// LS Electric XG5000 project: Master_UPH
// PLC LSPLC

PROGRAM NewProgram (task: Scan Program)

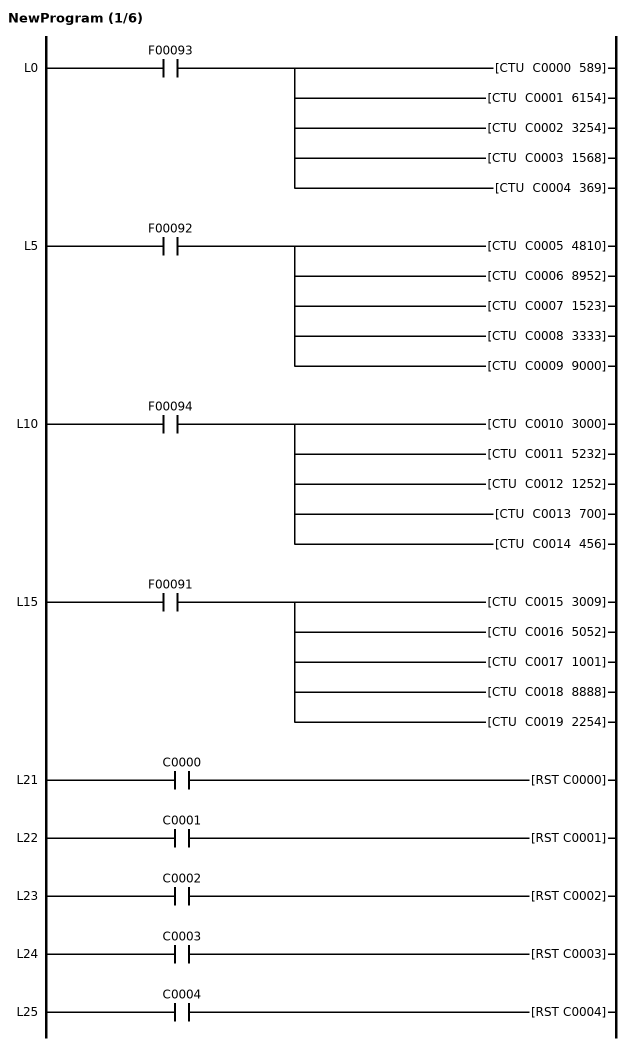
; L0
LOAD      F00093
CTU       C0000 589
CTU       C0001 6154
CTU       C0002 3254
CTU       C0003 1568
CTU       C0004 369
; L5
LOAD      F00092
CTU       C0005 4810
CTU       C0006 8952
CTU       C0007 1523
CTU       C0008 3333
CTU       C0009 9000
; L10
LOAD      F00094
CTU       C0010 3000
CTU       C0011 5232
CTU       C0012 1252
CTU       C0013 700
CTU       C0014 456
; L15
LOAD      F00091
CTU       C0015 3009
CTU       C0016 5052
CTU       C0017 1001
CTU       C0018 8888
CTU       C0019 2254
; L21
LOAD      C0000
RST       C0000
; L22
LOAD      C0001
RST       C0001
; L23
LOAD      C0002
RST       C0002
; L24
LOAD      C0003
RST       C0003
; L25
LOAD      C0004
RST       C0004

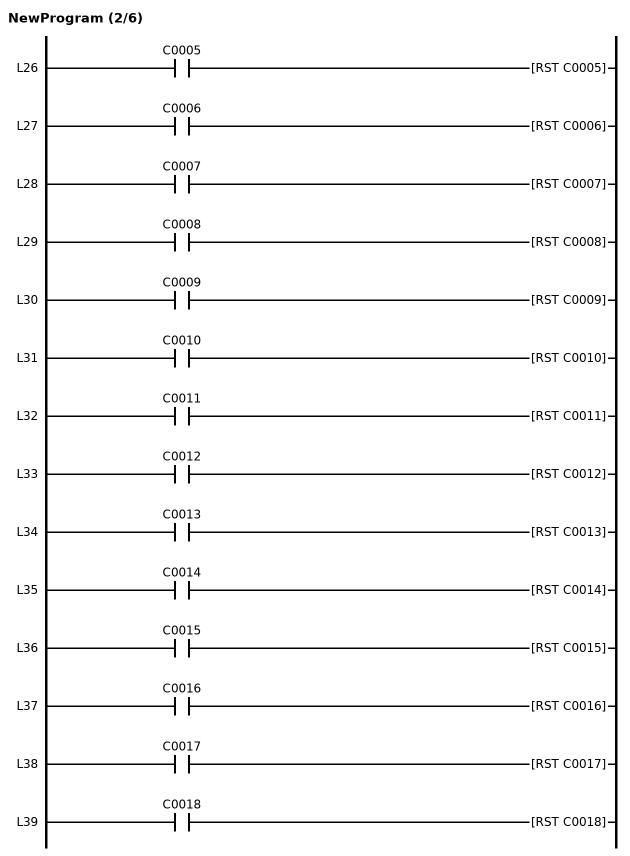
; L26
LOAD      C0005
RST       C0005
; L27
LOAD      C0006
RST       C0006
; L28
LOAD      C0007
RST       C0007
; L29
LOAD      C0008
RST       C0008
; L30
LOAD      C0009
RST       C0009
; L31
LOAD      C0010
RST       C0010
; L32
LOAD      C0011
RST       C0011
; L33
LOAD      C0012
RST       C0012
; L34
LOAD      C0013
RST       C0013
; L35
LOAD      C0014
RST       C0014
; L36
LOAD      C0015
RST       C0015
; L37
LOAD      C0016
RST       C0016
; L38
LOAD      C0017
RST       C0017
; L39
LOAD      C0018
RST       C0018

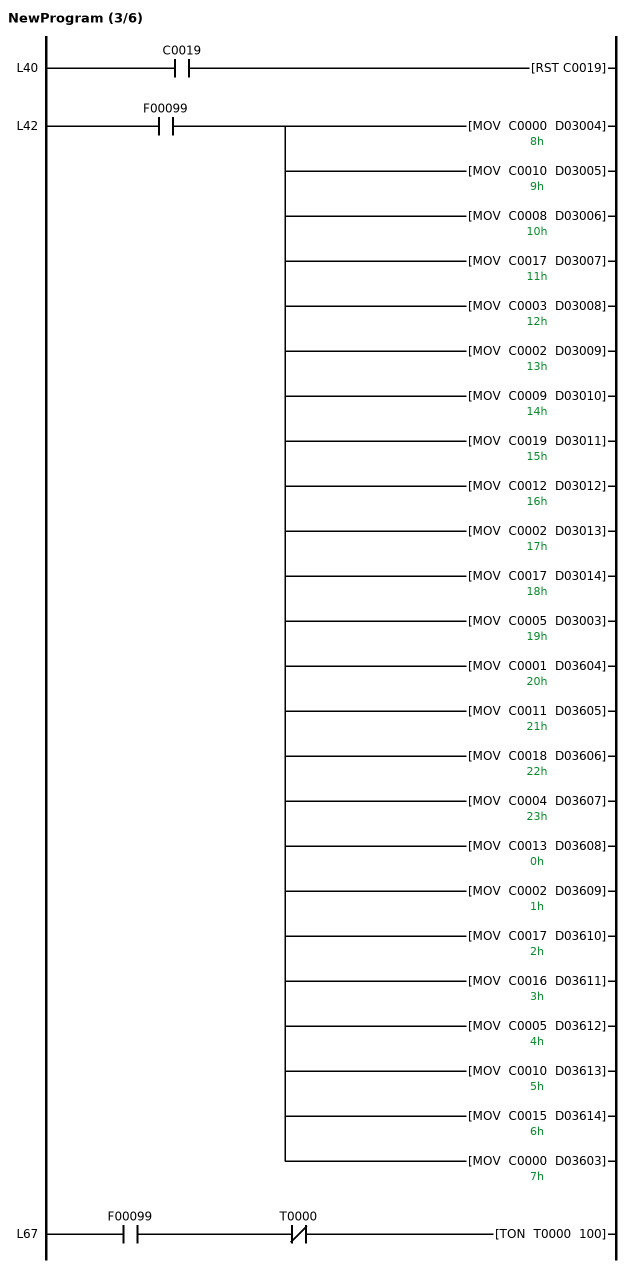
; L40
LOAD      C0019
RST       C0019
; L42
LOAD      F00099
MOV       C0000 D03004	// 8h
MOV       C0010 D03005	// 9h
MOV       C0008 D03006	// 10h
MOV       C0017 D03007	// 11h
MOV       C0003 D03008	// 12h
MOV       C0002 D03009	// 13h
MOV       C0009 D03010	// 14h
MOV       C0019 D03011	// 15h
MOV       C0012 D03012	// 16h
MOV       C0002 D03013	// 17h
MOV       C0017 D03014	// 18h
MOV       C0005 D03003	// 19h
MOV       C0001 D03604	// 20h
MOV       C0011 D03605	// 21h
MOV       C0018 D03606	// 22h
MOV       C0004 D03607	// 23h
MOV       C0013 D03608	// 0h
MOV       C0002 D03609	// 1h
MOV       C0017 D03610	// 2h
MOV       C0016 D03611	// 3h
MOV       C0005 D03612	// 4h
MOV       C0010 D03613	// 5h
MOV       C0015 D03614	// 6h
MOV       C0000 D03603	// 7h
; L67
LOAD      F00099
AND NOT   T0000
TON       T0000 100

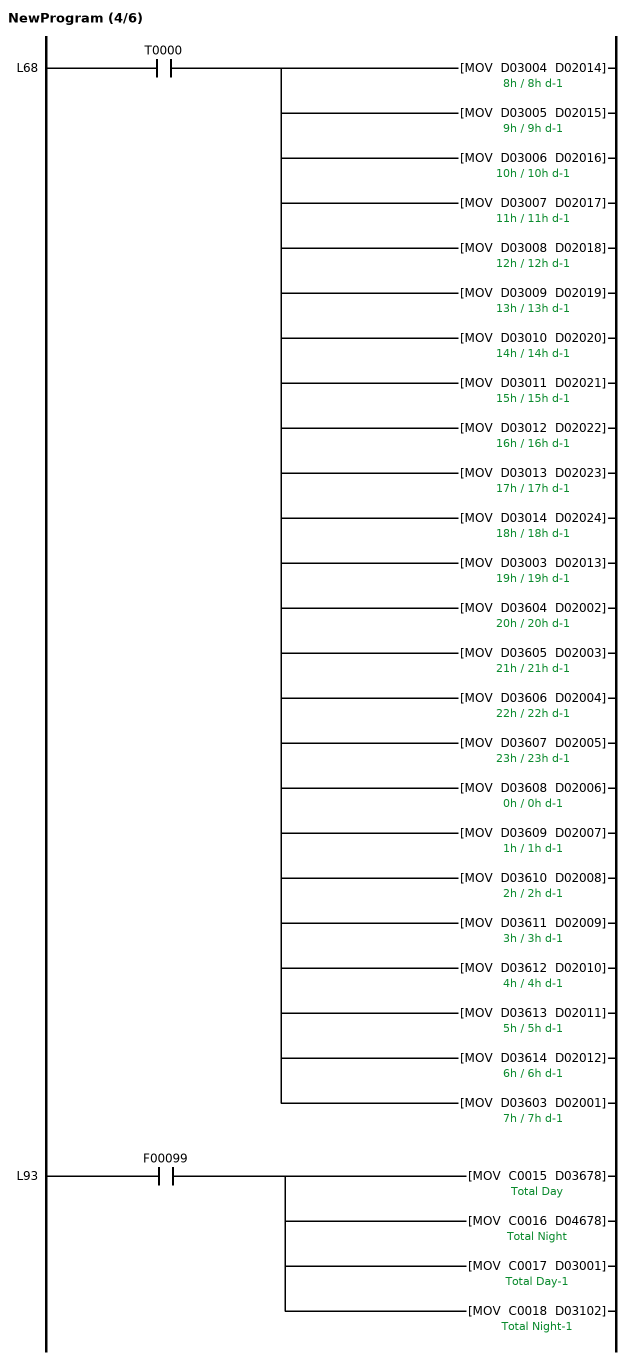
; L68
LOAD      T0000
MOV       D03004 D02014	// 8h / 8h d-1
MOV       D03005 D02015	// 9h / 9h d-1
MOV       D03006 D02016	// 10h / 10h d-1
MOV       D03007 D02017	// 11h / 11h d-1
MOV       D03008 D02018	// 12h / 12h d-1
MOV       D03009 D02019	// 13h / 13h d-1
MOV       D03010 D02020	// 14h / 14h d-1
MOV       D03011 D02021	// 15h / 15h d-1
MOV       D03012 D02022	// 16h / 16h d-1
MOV       D03013 D02023	// 17h / 17h d-1
MOV       D03014 D02024	// 18h / 18h d-1
MOV       D03003 D02013	// 19h / 19h d-1
MOV       D03604 D02002	// 20h / 20h d-1
MOV       D03605 D02003	// 21h / 21h d-1
MOV       D03606 D02004	// 22h / 22h d-1
MOV       D03607 D02005	// 23h / 23h d-1
MOV       D03608 D02006	// 0h / 0h d-1
MOV       D03609 D02007	// 1h / 1h d-1
MOV       D03610 D02008	// 2h / 2h d-1
MOV       D03611 D02009	// 3h / 3h d-1
MOV       D03612 D02010	// 4h / 4h d-1
MOV       D03613 D02011	// 5h / 5h d-1
MOV       D03614 D02012	// 6h / 6h d-1
MOV       D03603 D02001	// 7h / 7h d-1
; L93
LOAD      F00099
MOV       C0015 D03678	// Total Day
MOV       C0016 D04678	// Total Night
MOV       C0017 D03001	// Total Day-1
MOV       C0018 D03102	// Total Night-1

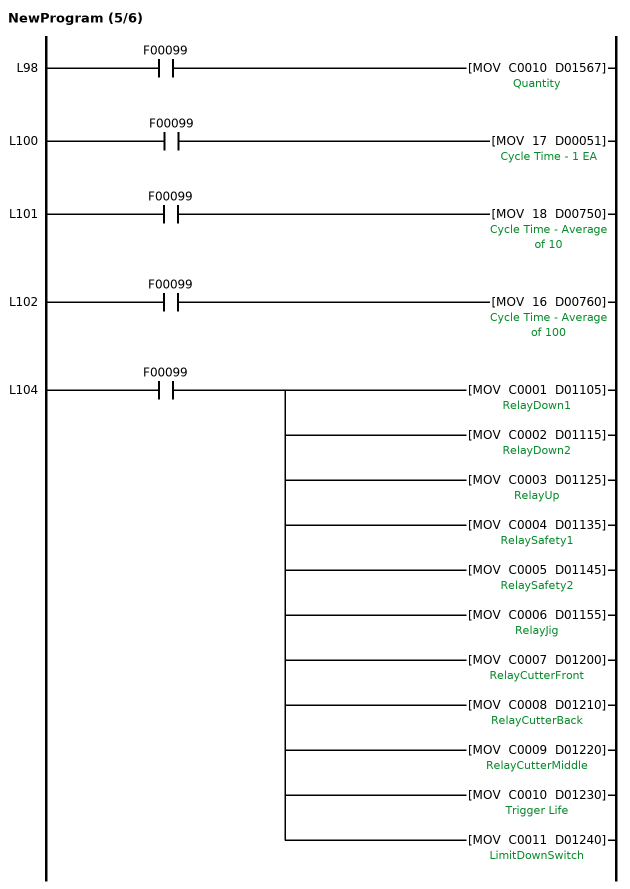
; L98
LOAD      F00099
MOV       C0010 D01567	// Quantity
; L100
LOAD      F00099
MOV       17 D00051	// Cycle Time - 1 EA
; L101
LOAD      F00099
MOV       18 D00750	// Cycle Time - Average of 10
; L102
LOAD      F00099
MOV       16 D00760	// Cycle Time - Average of 100
; L104
LOAD      F00099
MOV       C0001 D01105	// RelayDown1
MOV       C0002 D01115	// RelayDown2
MOV       C0003 D01125	// RelayUp
MOV       C0004 D01135	// RelaySafety1
MOV       C0005 D01145	// RelaySafety2
MOV       C0006 D01155	// RelayJig
MOV       C0007 D01200	// RelayCutterFront
MOV       C0008 D01210	// RelayCutterBack
MOV       C0009 D01220	// RelayCutterMiddle
MOV       C0010 D01230	// Trigger Life
MOV       C0011 D01240	// LimitDownSwitch

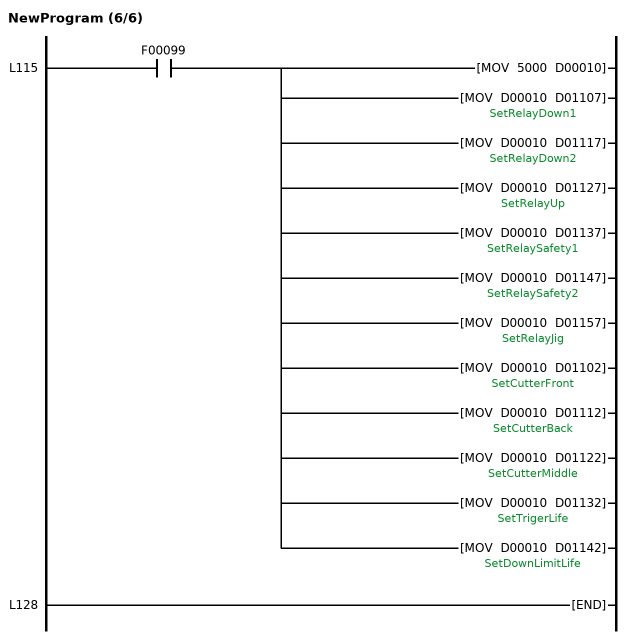
; L115
LOAD      F00099
MOV       5000 D00010
MOV       D00010 D01107	// SetRelayDown1
MOV       D00010 D01117	// SetRelayDown2
MOV       D00010 D01127	// SetRelayUp
MOV       D00010 D01137	// SetRelaySafety1
MOV       D00010 D01147	// SetRelaySafety2
MOV       D00010 D01157	// SetRelayJig
MOV       D00010 D01102	// SetCutterFront
MOV       D00010 D01112	// SetCutterBack
MOV       D00010 D01122	// SetCutterMiddle
MOV       D00010 D01132	// SetTrigerLife
MOV       D00010 D01142	// SetDownLimitLife
; L128
END

PROGRAM SQL (task: Scan Program)

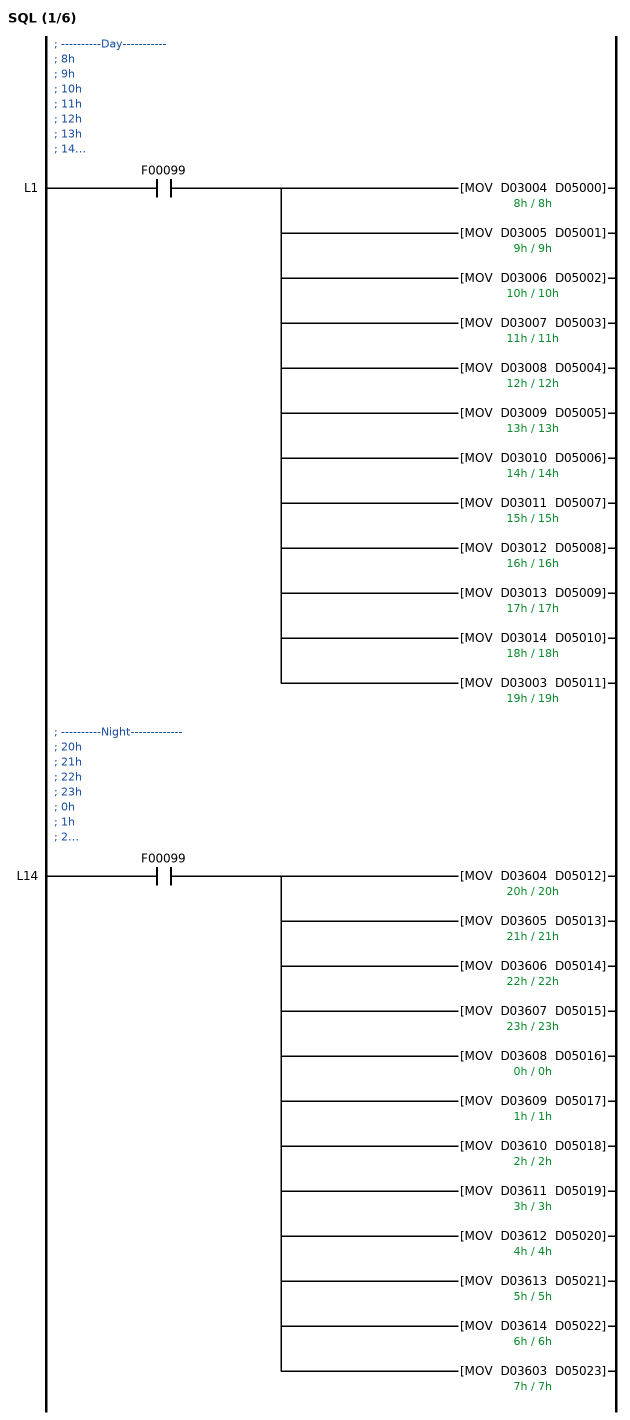
// ----------Day-----------
; L1
LOAD      F00099
MOV       D03004 D05000	// 8h / 8h
MOV       D03005 D05001	// 9h / 9h
MOV       D03006 D05002	// 10h / 10h
MOV       D03007 D05003	// 11h / 11h
MOV       D03008 D05004	// 12h / 12h
MOV       D03009 D05005	// 13h / 13h
MOV       D03010 D05006	// 14h / 14h
MOV       D03011 D05007	// 15h / 15h
MOV       D03012 D05008	// 16h / 16h
MOV       D03013 D05009	// 17h / 17h
MOV       D03014 D05010	// 18h / 18h
MOV       D03003 D05011	// 19h / 19h
// output comment: 8h
// output comment: 9h
// output comment: 10h
// output comment: 11h
// output comment: 12h
// output comment: 13h
// output comment: 14h
// output comment: 15h
// output comment: 16h
// output comment: 17h
// output comment: 18h
// output comment: 19h
// ----------Night-------------
; L14
LOAD      F00099
MOV       D03604 D05012	// 20h / 20h
MOV       D03605 D05013	// 21h / 21h
MOV       D03606 D05014	// 22h / 22h
MOV       D03607 D05015	// 23h / 23h
MOV       D03608 D05016	// 0h / 0h
MOV       D03609 D05017	// 1h / 1h
MOV       D03610 D05018	// 2h / 2h
MOV       D03611 D05019	// 3h / 3h
MOV       D03612 D05020	// 4h / 4h
MOV       D03613 D05021	// 5h / 5h
MOV       D03614 D05022	// 6h / 6h
MOV       D03603 D05023	// 7h / 7h
// output comment: 20h
// output comment: 21h
// output comment: 22h
// output comment: 23h
// output comment: 0h
// output comment: 1h
// output comment: 2h
// output comment: 3h
// output comment: 4h
// output comment: 5h
// output comment: 6h
// output comment: 7h

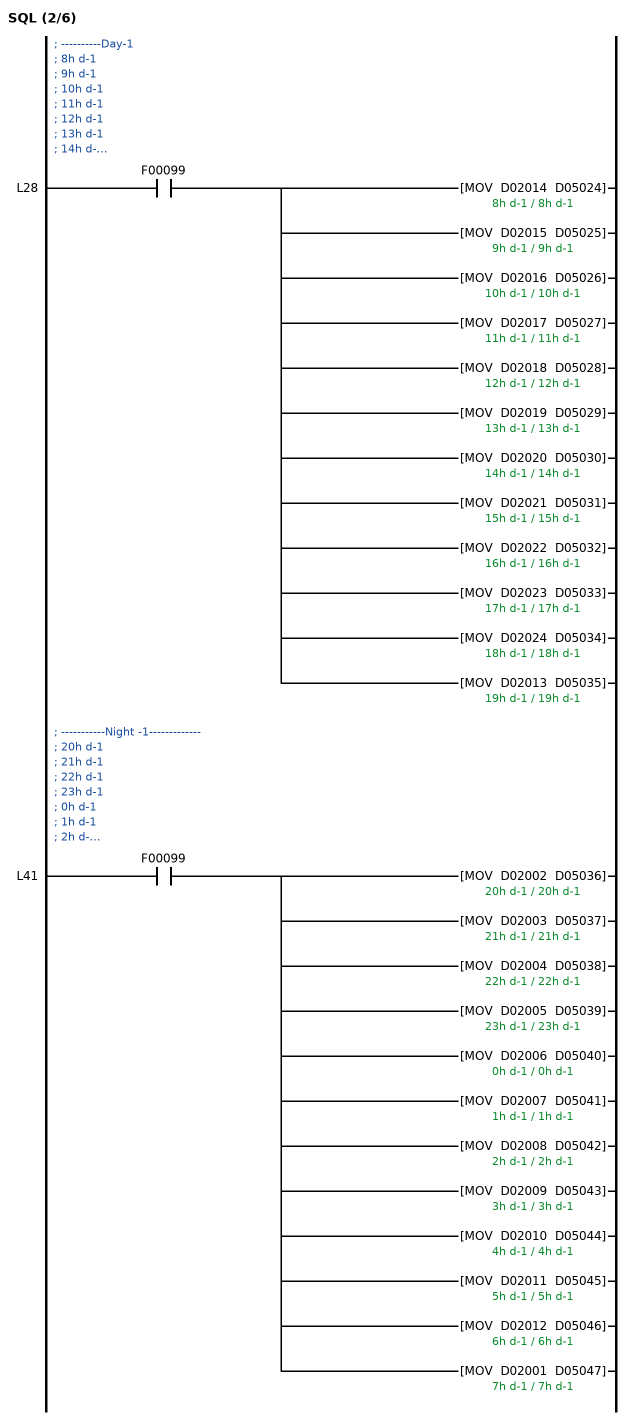
// ----------Day-1
; L28
LOAD      F00099
MOV       D02014 D05024	// 8h d-1 / 8h d-1
MOV       D02015 D05025	// 9h d-1 / 9h d-1
MOV       D02016 D05026	// 10h d-1 / 10h d-1
MOV       D02017 D05027	// 11h d-1 / 11h d-1
MOV       D02018 D05028	// 12h d-1 / 12h d-1
MOV       D02019 D05029	// 13h d-1 / 13h d-1
MOV       D02020 D05030	// 14h d-1 / 14h d-1
MOV       D02021 D05031	// 15h d-1 / 15h d-1
MOV       D02022 D05032	// 16h d-1 / 16h d-1
MOV       D02023 D05033	// 17h d-1 / 17h d-1
MOV       D02024 D05034	// 18h d-1 / 18h d-1
MOV       D02013 D05035	// 19h d-1 / 19h d-1
// output comment: 8h d-1
// output comment: 9h d-1
// output comment: 10h d-1
// output comment: 11h d-1
// output comment: 12h d-1
// output comment: 13h d-1
// output comment: 14h d-1
// output comment: 15h d-1
// output comment: 16h d-1
// output comment: 17h d-1
// output comment: 18h d-1
// output comment: 19h d-1
// -----------Night -1-------------
; L41
LOAD      F00099
MOV       D02002 D05036	// 20h d-1 / 20h d-1
MOV       D02003 D05037	// 21h d-1 / 21h d-1
MOV       D02004 D05038	// 22h d-1 / 22h d-1
MOV       D02005 D05039	// 23h d-1 / 23h d-1
MOV       D02006 D05040	// 0h d-1 / 0h d-1
MOV       D02007 D05041	// 1h d-1 / 1h d-1
MOV       D02008 D05042	// 2h d-1 / 2h d-1
MOV       D02009 D05043	// 3h d-1 / 3h d-1
MOV       D02010 D05044	// 4h d-1 / 4h d-1
MOV       D02011 D05045	// 5h d-1 / 5h d-1
MOV       D02012 D05046	// 6h d-1 / 6h d-1
MOV       D02001 D05047	// 7h d-1 / 7h d-1
// output comment: 20h d-1
// output comment: 21h d-1
// output comment: 22h d-1
// output comment: 23h d-1
// output comment: 0h d-1
// output comment: 1h d-1
// output comment: 2h d-1
// output comment: 3h d-1
// output comment: 4h d-1
// output comment: 5h d-1
// output comment: 6h d-1
// output comment: 7h d-1

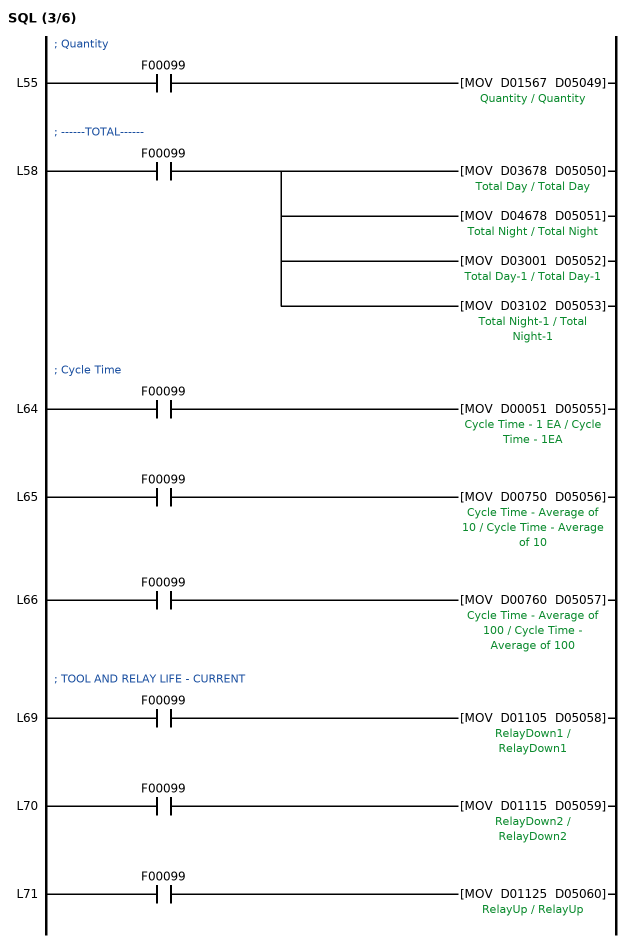
// Quantity
; L55
LOAD      F00099
MOV       D01567 D05049	// Quantity / Quantity
// ------TOTAL------
; L58
LOAD      F00099
MOV       D03678 D05050	// Total Day / Total Day
MOV       D04678 D05051	// Total Night / Total Night
MOV       D03001 D05052	// Total Day-1 / Total Day-1
MOV       D03102 D05053	// Total Night-1 / Total Night-1
// Cycle Time
; L64
LOAD      F00099
MOV       D00051 D05055	// Cycle Time - 1 EA / Cycle Time - 1EA
; L65
LOAD      F00099
MOV       D00750 D05056	// Cycle Time - Average of 10 / Cycle Time - Average of 10
; L66
LOAD      F00099
MOV       D00760 D05057	// Cycle Time - Average of 100 / Cycle Time - Average of 100
// TOOL AND RELAY LIFE - CURRENT
; L69
LOAD      F00099
MOV       D01105 D05058	// RelayDown1 / RelayDown1
; L70
LOAD      F00099
MOV       D01115 D05059	// RelayDown2 / RelayDown2
; L71
LOAD      F00099
MOV       D01125 D05060	// RelayUp / RelayUp

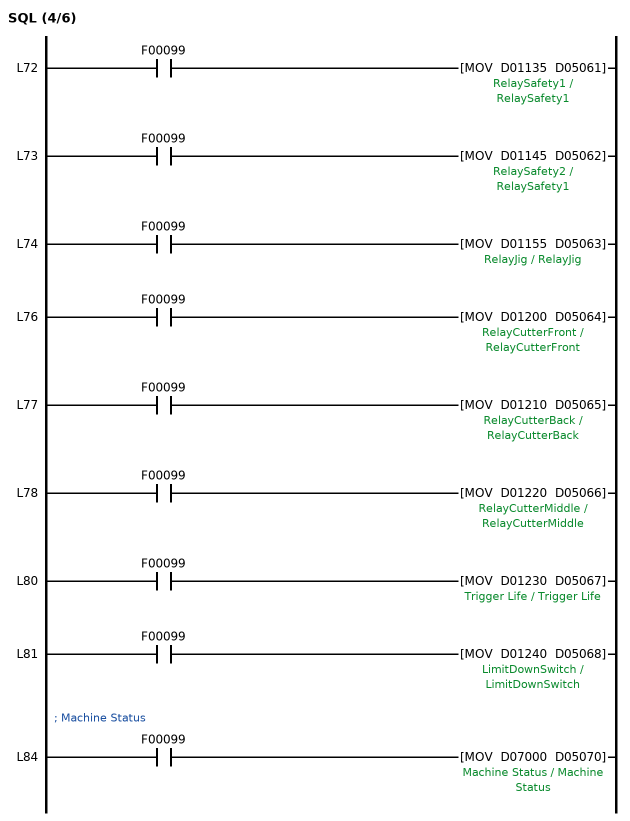
; L72
LOAD      F00099
MOV       D01135 D05061	// RelaySafety1 / RelaySafety1
; L73
LOAD      F00099
MOV       D01145 D05062	// RelaySafety2 / RelaySafety1
; L74
LOAD      F00099
MOV       D01155 D05063	// RelayJig / RelayJig
; L76
LOAD      F00099
MOV       D01200 D05064	// RelayCutterFront / RelayCutterFront
; L77
LOAD      F00099
MOV       D01210 D05065	// RelayCutterBack / RelayCutterBack
; L78
LOAD      F00099
MOV       D01220 D05066	// RelayCutterMiddle / RelayCutterMiddle
; L80
LOAD      F00099
MOV       D01230 D05067	// Trigger Life / Trigger Life
; L81
LOAD      F00099
MOV       D01240 D05068	// LimitDownSwitch / LimitDownSwitch
// Machine Status
; L84
LOAD      F00099
MOV       D07000 D05070	// Machine Status / Machine Status

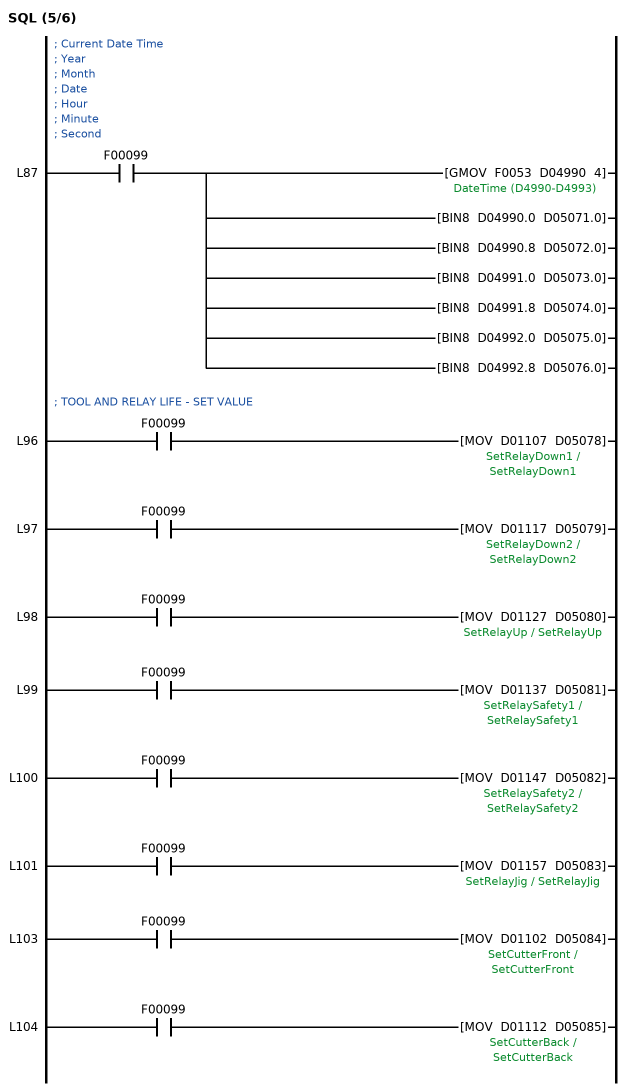
// Current Date Time
; L87
LOAD      F00099
GMOV      F0053 D04990 4	// DateTime (D4990-D4993)
BIN8      D04990.0 D05071.0
BIN8      D04990.8 D05072.0
BIN8      D04991.0 D05073.0
BIN8      D04991.8 D05074.0
BIN8      D04992.0 D05075.0
BIN8      D04992.8 D05076.0
// output comment: Year
// output comment: Month
// output comment: Date
// output comment: Hour
// output comment: Minute
// output comment: Second
// TOOL AND RELAY LIFE - SET VALUE
; L96
LOAD      F00099
MOV       D01107 D05078	// SetRelayDown1 / SetRelayDown1
; L97
LOAD      F00099
MOV       D01117 D05079	// SetRelayDown2 / SetRelayDown2
; L98
LOAD      F00099
MOV       D01127 D05080	// SetRelayUp / SetRelayUp
; L99
LOAD      F00099
MOV       D01137 D05081	// SetRelaySafety1 / SetRelaySafety1
; L100
LOAD      F00099
MOV       D01147 D05082	// SetRelaySafety2 / SetRelaySafety2
; L101
LOAD      F00099
MOV       D01157 D05083	// SetRelayJig / SetRelayJig
; L103
LOAD      F00099
MOV       D01102 D05084	// SetCutterFront / SetCutterFront
; L104
LOAD      F00099
MOV       D01112 D05085	// SetCutterBack / SetCutterBack

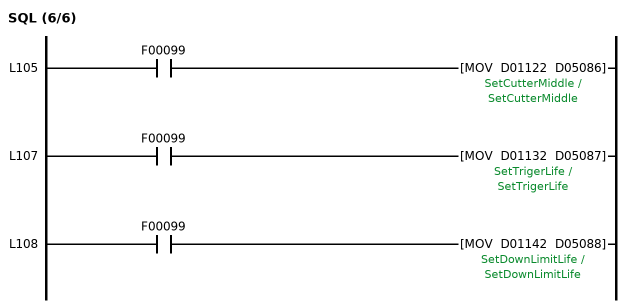
; L105
LOAD      F00099
MOV       D01122 D05086	// SetCutterMiddle / SetCutterMiddle
; L107
LOAD      F00099
MOV       D01132 D05087	// SetTrigerLife / SetTrigerLife
; L108
LOAD      F00099
MOV       D01142 D05088	// SetDownLimitLife / SetDownLimitLife

PROGRAM MachineStatus (task: Scan Program)

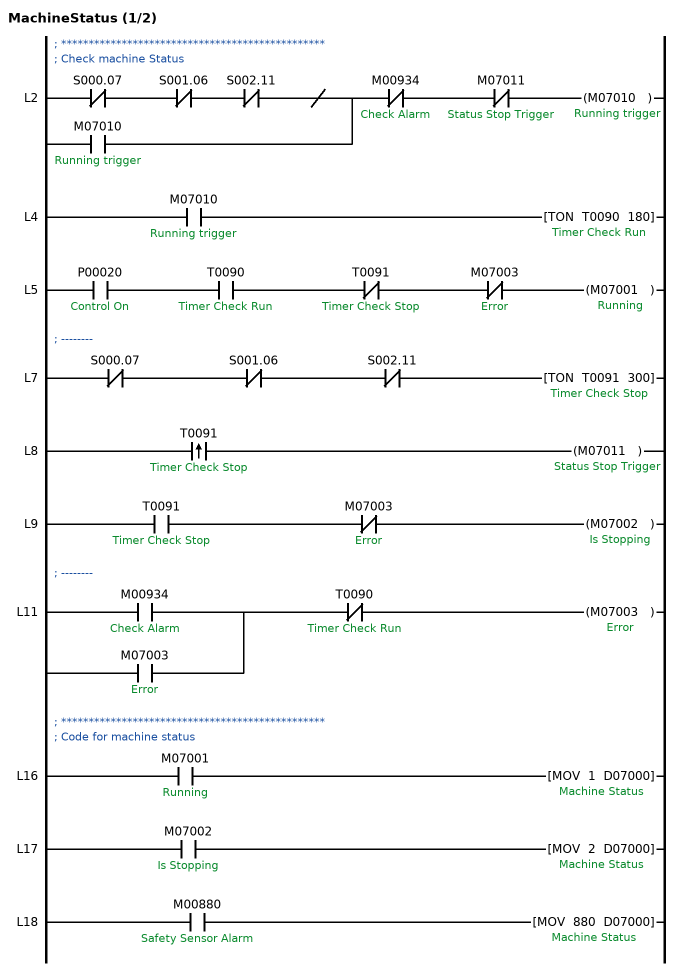
// ************************************************
// Check machine Status
; L2
LOAD NOT  S000.07
AND NOT   S001.06
AND NOT   S002.11
NOT
OR        M07010	// Running trigger
AND NOT   M00934	// Check Alarm
AND NOT   M07011	// Status Stop Trigger
OUT       M07010	// Running trigger
; L4
LOAD      M07010	// Running trigger
TON       T0090 180	// Timer Check Run
; L5
LOAD      P00020	// Control On
AND       T0090	// Timer Check Run
AND NOT   T0091	// Timer Check Stop
AND NOT   M07003	// Error
OUT       M07001	// Running
// --------
; L7
LOAD NOT  S000.07
AND NOT   S001.06
AND NOT   S002.11
TON       T0091 300	// Timer Check Stop
; L8
LOADP     T0091	// Timer Check Stop
OUT       M07011	// Status Stop Trigger
; L9
LOAD      T0091	// Timer Check Stop
AND NOT   M07003	// Error
OUT       M07002	// Is Stopping
// --------
; L11
LOAD      M00934	// Check Alarm
OR        M07003	// Error
AND NOT   T0090	// Timer Check Run
OUT       M07003	// Error
// ************************************************
// Code for machine status
; L16
LOAD      M07001	// Running
MOV       1 D07000	// Machine Status
; L17
LOAD      M07002	// Is Stopping
MOV       2 D07000	// Machine Status
; L18
LOAD      M00880	// Safety Sensor Alarm
MOV       880 D07000	// Machine Status

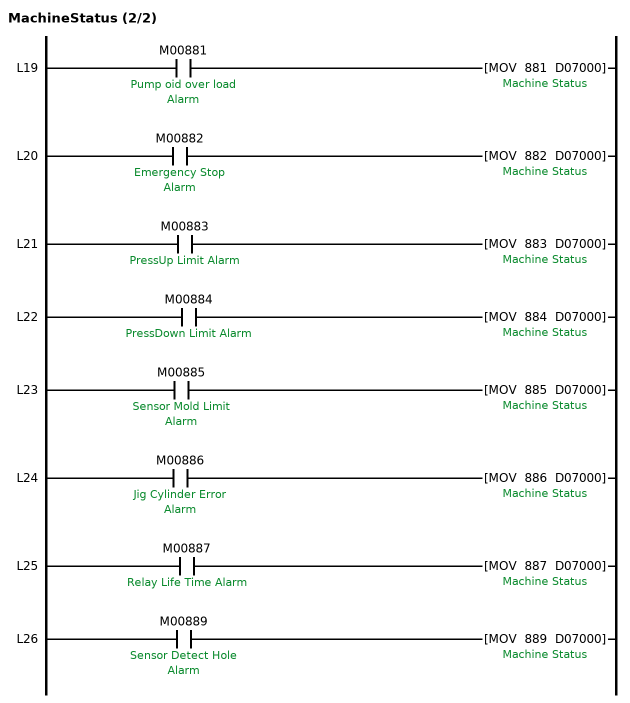
; L19
LOAD      M00881	// Pump oid over load Alarm
MOV       881 D07000	// Machine Status
; L20
LOAD      M00882	// Emergency Stop Alarm
MOV       882 D07000	// Machine Status
; L21
LOAD      M00883	// PressUp Limit Alarm
MOV       883 D07000	// Machine Status
; L22
LOAD      M00884	// PressDown Limit Alarm
MOV       884 D07000	// Machine Status
; L23
LOAD      M00885	// Sensor Mold Limit Alarm
MOV       885 D07000	// Machine Status
; L24
LOAD      M00886	// Jig Cylinder Error Alarm
MOV       886 D07000	// Machine Status
; L25
LOAD      M00887	// Relay Life Time Alarm
MOV       887 D07000	// Machine Status
; L26
LOAD      M00889	// Sensor Detect Hole Alarm
MOV       889 D07000	// Machine Status

VARIABLES AND COMMENTS (devices not used above)
M00301	BIT	CtrolOn_Light
S00007	BIT	Last Step A Mode
S00106	BIT	Last Step B Mode
S00211	BIT	Last Step C Mode